FUNCTION_BLOCK FB_Evt_Misc EXTENDS FB_BA_View
VAR
	{region 'Iteration'}
		// Intention:			Iterate over active events.
		bIterate				: BOOL;
		bIterate_ShowTimestamp	: BOOL				:= FALSE;
		bIterate_ShowType		: BOOL				:= TRUE;
		bIterate_ShowState		: BOOL				:= TRUE;
		bIterate_ShowEC			: BOOL				:= FALSE;
	{endregion}
END_VAR
VAR
	_i							: DINT;
	_sVal						: T_MaxString;
	_iObj						: I_BA_EventObject;
	_fbMsg						: FB_BA_DecorString;
END_VAR

SUPER^();

IF (bIterate) THEN
	bIterate := FALSE;
	
	_i := F_BA_GetEventCount();
	IF (_i = 0) THEN
		F_BA_LogMessage(ADSLOG_MSGTYPE_HINT, 'EM06', 'No active events found yet.');
	ELSE
		F_BA_LogMessage1(ADSLOG_MSGTYPE_HINT, 'EM08', 'Active events: %d', F_DINT(_i));
		
		// Iterate over all active events:
		_i := 0;
		_iObj := 0;								// [Hint] Temporary iterator-object must be NULL to start iteration from the beginning.
		WHILE (F_BA_IterateEvents(_iObj)) DO
			_i := (_i+1);
			
			// Format message:
			_fbMsg.Reset();
			IF (bIterate_ShowTimestamp) THEN
				_sVal := TO_STRING(F_BA_ToDT(_iObj.EventChangeTime));
				_fbMsg.AddDecor1('%s', F_STRING(_sVal));
			END_IF
			IF (bIterate_ShowType) THEN
				_fbMsg.AddDecor1('Type: %s', F_STRINGEx(BA_EnumEN.aEventType[_iObj.EventIcon.eEventType].sName));
			END_IF
			IF (bIterate_ShowState) THEN
				_fbMsg.AddDecor1('State: %s', F_STRINGEx(BA_EnumEN.aEventIconState[_iObj.EventIcon.eState].sDescription));
			END_IF
			IF (bIterate_ShowEC) THEN
				_sVal := TO_STRING(_iObj.EventClassID);
				_fbMsg.AddDecor1('Event class: %s', F_STRING(_sVal));
			END_IF
			_fbMsg.Finish();
			
			_sVal := _iObj.ObjectName;
			F_BA_LogMessage3(ADSLOG_MSGTYPE_HINT, 'EM32', '%d. %s   %s', F_DINT(_i), F_STRING(_sVal), F_STRING(_fbMsg.sOutput));
		END_WHILE
	END_IF
END_IF

END_FUNCTION_BLOCK

(* stored: Version 1.1.0.1, ProductVersion 3.1.4024.11
   POU FB_Evt_Misc: Id {fe5b2e62-a31c-4ee5-b1db-d4befbe56498}, SpecialFunc None *)
